FUNCTION_BLOCK FB_2_AlimentarBase_SFC
VAR_INPUT
	
	//  SFC-Flags
	SFCPause: BOOL;
	SFCReset: BOOL;

	// Indicadores de sincronización
	Ack: BOOL := TRUE;
	Execute: BOOL;
	
	// Entradas
	AlimentadorDetras: BOOL;
	AlimentadorDelante: BOOL;
	PresenciaBaseAlimentador: BOOL;
	PulsadorMarcha: BOOL;
	
END_VAR
VAR_OUTPUT
	
	// Indicadores de sincronización
	Ready: BOOL;	
	Done: BOOL;
	
	// Salidas
	AlimentadorAdelante: BOOL;
	LamparaFaltaMaterial: BOOL;
	
END_VAR
VAR
END_VAR

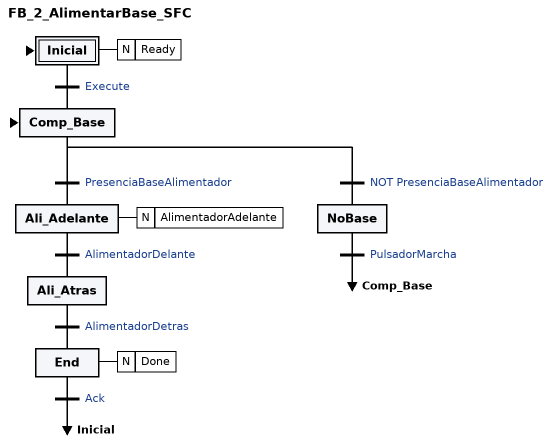
INITIAL_STEP Inicial:
    Ready(N);
END_STEP
TRANSITION FROM Inicial TO Comp_Base
    := Execute;
END_TRANSITION
STEP Comp_Base:
END_STEP
TRANSITION FROM Comp_Base TO Ali_Adelante
    := PresenciaBaseAlimentador;
END_TRANSITION
TRANSITION FROM Comp_Base TO NoBase
    := NOT PresenciaBaseAlimentador;
END_TRANSITION
STEP NoBase:
END_STEP
TRANSITION FROM NoBase TO Comp_Base
    := PulsadorMarcha;
END_TRANSITION
STEP Ali_Adelante:
    AlimentadorAdelante(N);
END_STEP
TRANSITION FROM Ali_Adelante TO Ali_Atras
    := AlimentadorDelante;
END_TRANSITION
STEP Ali_Atras:
END_STEP
TRANSITION FROM Ali_Atras TO End
    := AlimentadorDetras;
END_TRANSITION
STEP End:
    Done(N);
END_STEP
TRANSITION FROM End TO Inicial
    := Ack;
END_TRANSITION

END_FUNCTION_BLOCK

(* stored: Version 1.1.0.1, ProductVersion 3.1.4024.12
   POU FB_2_AlimentarBase_SFC: Id {9aefa8c8-ac12-4791-909e-6a9e8a71434b}, SpecialFunc None *)
